//essa linha se aplica para os 2
//significa que passou a fila toda e nao encontrou onde largar entao provavelmente deu problema
IF i > 10 THEN
	xLimpaFilaTAG := TRUE;
END_IF

//limpa a fila de TAG
IF xLimpaFilaTAG THEN
	xLimpaFilaTAG := FALSE;
	FOR i := 0 TO 10 DO
		iFilaTAG[i] := 0;
	END_FOR
END_IF
END_ACTION

END_FUNCTION_BLOCK

// POUs/Automatico/Aspercao/RFIDeBalanca/FB_RFIDBalancaEntrada
FUNCTION_BLOCK FB_RFIDBalancaEntrada
VAR_INPUT
	xChegou : BOOL;//sinal de que uma carcaça chegou
	
	rPeso : REAL;//peso que veio da balanca
	xNovoPeso : BOOL;//sinal de que veio um novo peso
	
	iTAG : INT;//tag que veio da leitor
	xNovaTAG : BOOL;//sinal de que veio um novo tag
	
	iCamaraSelecionada : INT;//camara selecionada
	stHoraAhora 	: TIMESTRUCT; //Hora atual 
	sProcesso : STRING;//GUID do processo atual da camara que ele selecionou
	xLimpaFilaPeso : BOOL;
	xLimpaFilaTAG : BOOL;
END_VAR
VAR_OUTPUT
	iFilaTAG : ARRAY[0..10] OF INT;//fila das tag
	rFilaPeso : ARRAY[0..10] OF REAL;//fila dos pesos
	
	xEsperandoBalanca : BOOL;//se ta esperando vim o peso da balanca
	xEsperandoRFID : BOOL;//se ta esperando vim o valor da tag
	
	rPesoSelecionado : REAL;//qual peso ele selecionou e vai mandar para o banco
	iTAGSelecionado : INT;//qual tag ele selecionou e vai mandar para o banco
	
	stBuffer : ARRAY[0..9] OF st_BufferTagBalanca;
	
END_VAR
VAR
	i : INT;
	j : INT;
	rtChegouPeso : R_TRIG;
	rtTiraPeso : R_TRIG;
	xTiraPeso : BOOL;
	rtChegouTAG : R_TRIG;
	rtTiraTAG : R_TRIG;
	xTiraTAG : BOOL;
	
	rtChegou : R_TRIG;
	
	iEstado : INT;
	
						
	sSB		  : FB_StringBuilder;
    fbPLCDBCmd    : FB_PLCDBCmdEvt(sNetID := '', tTimeout := T#5S);
    sCmd          : STRING (1000); 
    aPara         : ST_ExpParameter;
	sAux 		  : STRING;
	
	stTSAux 	  : TIMESTRUCT; //Hora atual 
	
	
	saAux : ARRAY[0..50] OF STRING(80);//para gerar os comandos
	
END_VAR



IF true THEN	

	ControlePeso();
	ControleTAG();
	
	
	rtChegou(CLK:= xNovaTAG OR xChegou, Q=> );
	
	
	CASE  iEstado OF 
		0://esperando chegar 
			IF rtChegou.Q THEN
				xEsperandoBalanca := TRUE;
				xEsperandoRFID := TRUE;
				iEstado := 1;
			END_IF
			
		1://chegou fica esperando ter alguma 
				
			xEsperandoRFID := iFilaTAG[0] = 0;
			xEsperandoBalanca := rFilaPeso[0] = 0;
			
			IF NOT xEsperandoRFID AND NOT xEsperandoBalanca THEN
				iEstado := 2;
				rPesoSelecionado := rFilaPeso[0];
				xTiraPeso := TRUE;
				xEsperandoBalanca := FALSE;
				
				iTAGSelecionado := iFilaTAG[0];
				xTiraTAG := TRUE;
				xEsperandoRFID := FALSE;
				
				iEstado := 2;
				
				//ajusta no buffer
				FOR i := 9 TO 1 BY -1 DO
					stBuffer[i] := stBuffer[i-1];
				END_FOR
				
				stBuffer[0].iTag := iTAGSelecionado;
				stBuffer[0].rPeso := rPesoSelecionado;
				
				
			END_IF
		
		2://manda pro banco esses valores
		
			FOR i:= 0 TO 50 DO
				saAux[i] := '';
			END_FOR
			
			saAux[0] := ('INSERT INTO `geral`.`rfid` (`TAG`, `Processo`, ');
			saAux[1] := ('`Camara`, `PesoQuente`, `HoraPesoQuente`) VALUES ($'');
			saAux[2] := (TO_STRING(iTAGSelecionado));
			saAux[3] := ('$', $'');
			saAux[4] := (TO_STRING(sProcesso));
			saAux[5] := ('$', $'');
			saAux[6] := (TO_STRING(iCamaraSelecionada));
			saAux[7] := ('$', $'');
			saAux[8] := (TO_STRING(rPesoSelecionado));
			saAux[9] := ('$', $'');
			saAux[10] := (TO_STRING(stHoraAhora.wYear));
			saAux[11] := ('-');
			saAux[13] := (TO_STRING(stHoraAhora.wMonth));
			saAux[14] := ('-');
			saAux[15] := (TO_STRING(stHoraAhora.wDay));
			saAux[16] := (' ');
			saAux[17] := (TO_STRING(stHoraAhora.wHour));
			saAux[18] := (':');
			saAux[19] := (TO_STRING(stHoraAhora.wMinute));
			saAux[20] := (':');
			saAux[21] := (TO_STRING(stHoraAhora.wSecond));
			saAux[22] := ('$');');
			
			sCmd := F_ConcatArray1000(sArray:= saAux);
			
			aPara.eParaType := E_ExpParameterType.STRING_;
			aPara.nParaSize := SIZEOF(sAux);
		
			// call functionblock
			IF fbPLCDBCmd.Execute(
				hDBID:= 1, 
				pExpression:= ADR(sCmd), 
				cbExpression:= SIZEOF(sCmd), 
				pData:= ADR(sAux), 
				cbData:= SIZEOF(sAux), 
				pParameter:= ADR(aPara), 
				cbParameter:= SIZEOF(aPara)) 
			THEN
				iEstado := 0;
			END_IF
		
	END_CASE
	


END_IF

ACTION ControlePeso:



//Sobe na fila
rtChegouPeso(CLK:= xNovoPeso AND xEsperandoBalanca, Q=> );
IF rtChegouPeso.q THEN
	FOR i := 0 TO 9 DO
		IF rFilaPeso[i] = 0 THEN
			rFilaPeso[i] := rPeso;
			EXIT;
		END_IF
	END_FOR
END_IF


//Sobe na fila
rtTiraPeso(CLK:= xTiraPeso, Q=> );
IF rtTiraPeso.q THEN
	xTiraPeso := false;
	FOR i := 0 TO 9 DO
		IF rFilaPeso[i] = 0 THEN
			FOR j := 0 TO i DO
				rFilaPeso[j] := rFilaPeso[j+1];
			END_FOR
			EXIT;
		END_IF
	END_FOR
END_IF

//essa linha se aplica para os 2
//significa que passou a fila toda e nao encontrou onde largar entao provavelmente deu problema
IF i > 10 THEN
	xLimpaFilaPeso := TRUE;
END_IF

//limpa a fila de peso
IF xLimpaFilaPeso THEN
	xLimpaFilaPeso := FALSE;
	FOR i := 0 TO 10 DO
		rFilaPeso[i] := 0;
	END_FOR
END_IF
END_ACTION

ACTION ControleTAG:


//Sobe na fila
rtChegouTAG(CLK:= xNovaTAG, Q=> );
IF rtChegouTAG.q THEN
	FOR i := 0 TO 9 DO
		IF iFilaTAG[i] = 0 THEN
			iFilaTAG[i] := iTAG;
			EXIT;
		END_IF
	END_FOR
END_IF


//Sobe na fila
rtTiraTAG(CLK:= xTiraTAG, Q=> );
IF rtTiraTAG.q THEN
	xTiraTAG := false;
	FOR i := 0 TO 9 DO
		IF iFilaTAG[i] = 0 THEN
			FOR j := 0 TO i DO
				iFilaTAG[j] := iFilaTAG[j+1];
			END_FOR
			EXIT;
		END_IF
	END_FOR
END_IF

//essa linha se aplica para os 2
//significa que passou a fila toda e nao encontrou onde largar entao provavelmente deu problema
IF i > 10 THEN
	xLimpaFilaTAG := TRUE;
END_IF

//limpa a fila de TAG
IF xLimpaFilaTAG THEN
	xLimpaFilaTAG := FALSE;
	FOR i := 0 TO 10 DO
		iFilaTAG[i] := 0;
	END_FOR
END_IF
END_ACTION

END_FUNCTION_BLOCK

// POUs/Automatico/Aspercao/RFIDeBalanca/FB_RFIDBalancaSaida
FUNCTION_BLOCK FB_RFIDBalancaSaida
VAR_INPUT
	xChegou : BOOL;
	
	rPeso : REAL;
	xNovoPeso : BOOL;
	
	iTAG : INT;
	xNovaTAG : BOOL;
	
	iCamaraSelecionada : INT;
	stHoraAhora 	: TIMESTRUCT; //Hora atual 
	sProcesso : STRING;
	xLimpaFilaPeso : BOOL;
	xLimpaFilaTAG : BOOL;
	
END_VAR
VAR_OUTPUT
	iFilaTAG : ARRAY[0..10] OF INT;
	rFilaPeso : ARRAY[0..10] OF REAL;
	
	xEsperandoBalanca : BOOL;
	xEsperandoRFID : BOOL;
	
	rPesoSelecionado : REAL;
	iTAGSelecionado : INT;
	
	
	stBuffer : ARRAY[0..9] OF st_BufferTagBalanca;
	
END_VAR
VAR
	i : INT;
	j : INT;
	rtChegouPeso : R_TRIG;
	rtTiraPeso : R_TRIG;
	xTiraPeso : BOOL;
	rtChegouTAG : R_TRIG;
	rtTiraTAG : R_TRIG;
	xTiraTAG : BOOL;
	
	rtChegou : R_TRIG;
	
	iEstado : INT;
	
						
	//sSB		  : FB_StringBuilder;
    fbPLCDBCmd    : FB_PLCDBCmdEvt(sNetID := '', tTimeout := T#5S);
    sCmd          : STRING (1000); 
    aPara         : ST_ExpParameter;
	sAux 		  : STRING;
	
	stTSAux 	  : TIMESTRUCT; //Hora atual 
	
	saAux : ARRAY[0..50] OF STRING(80);//para gerar os comandos
	
	
END_VAR



IF true THEN	

	ControlePeso();
	ControleTAG();
	
	
	rtChegou(CLK:= xNovaTAG OR xChegou, Q=> );
	
	CASE  iEstado OF 
		0://esperando chegar 
			IF rtChegou.q THEN
				xEsperandoBalanca := TRUE;
				xEsperandoRFID := TRUE;
				iEstado := 1;
			END_IF
			
		1://chegou fica esperando ter alguma 
				
			xEsperandoRFID := iFilaTAG[0] = 0;
			xEsperandoBalanca := rFilaPeso[0] = 0;
			
			IF NOT xEsperandoRFID AND NOT xEsperandoBalanca THEN
				iEstado := 2;
				rPesoSelecionado := rFilaPeso[0];
				xTiraPeso := TRUE;
				xEsperandoBalanca := FALSE;
				
				iTAGSelecionado := iFilaTAG[0];
				xTiraTAG := TRUE;
				xEsperandoRFID := FALSE;
				
				iEstado := 2;
				
				//ajusta no buffer
				FOR i := 9 TO 1 BY -1 DO
					stBuffer[i] := stBuffer[i-1];
				END_FOR
				
				stBuffer[0].iTag := iTAGSelecionado;
				stBuffer[0].rPeso := rPesoSelecionado;
				
				
			END_IF
		
		2://manda pro banco esses valores
			//UPDATE `geral`.`rfid` SET `PesoFrio` = '12', `HoraPesoFrio` = 'xxx' WHERE (`TAG` = '12' and `Processo` = '{28F6E224-5F99-464E-8EF2-4966F1D308DE}');
			
			FOR i:= 0 TO 50 DO
				saAux[i] := '';
			END_FOR
			
			saAux[0] := ('UPDATE `geral`.`rfid` SET `PesoFrio` = $'');
			saAux[1] := (TO_STRING(rPesoSelecionado));
			saAux[2] := ('$', `Camara` = $'');
			saAux[3] := (TO_STRING(iCamaraSelecionada));
			saAux[4] := ('$', `HoraPesoFrio` = $'');
			saAux[5] := (TO_STRING(stHoraAhora.wYear));
			saAux[6] := ('-');
			saAux[7] := (TO_STRING(stHoraAhora.wMonth));
			saAux[8] := ('-');
			saAux[9] := (TO_STRING(stHoraAhora.wDay));
			saAux[10] := (' ');
			saAux[11] := (TO_STRING(stHoraAhora.wHour));
			saAux[12] := (':');
			saAux[13] := (TO_STRING(stHoraAhora.wMinute));
			saAux[14] := (':');
			saAux[15] := (TO_STRING(stHoraAhora.wSecond));
			saAux[16] := ('$' WHERE (`TAG` = $'');
			saAux[17] := (TO_STRING(iTAG));
			saAux[18] := ('$' and `PesoFrio` = $'');
			saAux[19] := ('-1');
			saAux[20] := ('$'');
			saAux[21] := ('');
			saAux[22] := (') ORDER BY id DESC LIMIT 1;');
			// PesoFrio` = '-1' and DATE(`HoraPesoQuente`) = DATE(DATE_ADD(now(), INTERVAL -1 DAY))) ORDER BY id DESC LIMIT 1;
			
			sCmd := F_ConcatArray1000(sArray:= saAux);
			
			aPara.eParaType := E_ExpParameterType.STRING_;
			aPara.nParaSize := SIZEOF(sAux);
		
			// call functionblock
			IF fbPLCDBCmd.Execute(
				hDBID:= 1, 
				pExpression:= ADR(sCmd), 
				cbExpression:= SIZEOF(sCmd), 
				pData:= ADR(sAux), 
				cbData:= SIZEOF(sAux), 
				pParameter:= ADR(aPara), 
				cbParameter:= SIZEOF(aPara)) 
			THEN
				iEstado := 0;
			END_IF
		
	END_CASE
	
	
	
	



END_IF

ACTION ControlePeso:



//Sobe na fila
rtChegouPeso(CLK:= xNovoPeso AND xEsperandoBalanca, Q=> );
IF rtChegouPeso.q THEN
	FOR i := 0 TO 9 DO
		IF rFilaPeso[i] = 0 THEN
			rFilaPeso[i] := rPeso;
			EXIT;
		END_IF
	END_FOR
END_IF


//Sobe na fila
rtTiraPeso(CLK:= xTiraPeso, Q=> );
IF rtTiraPeso.q THEN
	xTiraPeso := false;
	FOR i := 0 TO 9 DO
		IF rFilaPeso[i] = 0 THEN
			FOR j := 0 TO i DO
				rFilaPeso[j] := rFilaPeso[j+1];
			END_FOR
			EXIT;
		END_IF
	END_FOR
END_IF

//essa linha se aplica para os 2
//significa que passou a fila toda e nao encontrou onde largar entao provavelmente deu problema
IF i > 10 THEN
	xLimpaFilaPeso := TRUE;
END_IF

//limpa a fila de peso
IF xLimpaFilaPeso THEN
	xLimpaFilaPeso := FALSE;
	FOR i := 0 TO 10 DO
		rFilaPeso[i] := 0;
	END_FOR
END_IF
END_ACTION

ACTION ControleTAG:


//Sobe na fila
rtChegouTAG(CLK:= xNovaTAG, Q=> );
IF rtChegouTAG.q THEN
	FOR i := 0 TO 9 DO
		IF iFilaTAG[i] = 0 THEN
			iFilaTAG[i] := iTAG;
			EXIT;
		END_IF
	END_FOR
END_IF


//Sobe na fila
rtTiraTAG(CLK:= xTiraTAG, Q=> );
IF rtTiraTAG.q THEN
	xTiraTAG := false;
	FOR i := 0 TO 9 DO
		IF iFilaTAG[i] = 0 THEN
			FOR j := 0 TO i DO
				iFilaTAG[j] := iFilaTAG[j+1];
			END_FOR
			EXIT;
		END_IF
	END_FOR
END_IF

//essa linha se aplica para os 2
//significa que passou a fila toda e nao encontrou onde largar entao provavelmente deu problema
IF i > 10 THEN
	xLimpaFilaTAG := TRUE;
END_IF

//limpa a fila de TAG
IF xLimpaFilaTAG THEN
	xLimpaFilaTAG := FALSE;
	FOR i := 0 TO 10 DO
		iFilaTAG[i] := 0;
	END_FOR
END_IF
END_ACTION

END_FUNCTION_BLOCK

// POUs/Automatico/ControlesPID/FB_PIDeGrafico
FUNCTION_BLOCK FB_PIDeGrafico
VAR_IN_OUT
	stPID : stControlePID;
END_VAR
VAR_OUTPUT
END_VAR
VAR
	PID : FB_CTRL_PID;
	tonTempoDeAmostragem : TON;
	i : INT;
END_VAR





stPID.PID.EN.fSetpointValue := stPID.Config.rSetpoint;//Setpoint
stPID.PID.EN.fActualValue;//Valor atual
stPID.PID.EN.fManSyncValue;//Valor em manual
IF stPID.xLigaInterno THEN
	stPID.PID.EN.eMode := eCTRL_MODE_ACTIVE;
ELSE
	stPID.PID.EN.eMode := eCTRL_MODE_PASSIVE;	
END_IF
IF stPID.xReset THEN
	stPID.PID.EN.eMode := eCTRL_MODE_RESET;
END_IF
//eCTRL_MODE_PASSIVE - The output or outputs of the function block are set to zero, but the internal states are retained.
//eCTRL_MODE_ACTIVE - The function block is executed in accordance with its description, and appropriate output values are calculated (normal operation).
//eCTRL_MODE_RESET - In this operation mode all internal states are reset and the error bit is cleared.
//eCTRL_MODE_MANUAL - The value of the input value fManSyncValue is provided at the output (manual operation).
//eCTRL_STATE_IDLE - The function block has successfully been reset, and is now waiting for selection of the operation mode.


stPID.PID.stParams.tTaskCycleTime := T#10MS;//Tempo igual ao da Task PID
stPID.PID.stParams.tCtrlCycleTime := T#50MS;//A cada quanto tempo vai rodar o bloco

stPID.PID.stParams.fKp;//Controller amplification / controller coefficient
stPID.PID.stParams.tTn;//Integral action time; if this is parameterized to T#0s, the I component is deactivated.
stPID.PID.stParams.tTv;//Derivative action time; if this is parameterized to T#0s, the D component is deactivated.
stPID.PID.stParams.tTd;//Damping time
IF stPID.xPressao THEN
	stPID.PID.stParams.fOutMaxLimit := 100;
	stPID.PID.stParams.fOutMinLimit := 0;
ELSE
	stPID.PID.stParams.fOutMaxLimit := 100;
	stPID.PID.stParams.fOutMinLimit := 0;	
END_IF

aPID();

IF stPID.xPressao THEN
	stPID.PID.SA.rSaida := SCALE_R(X := stPID.PID.SA.fOut,
											I_LO := 0,
											I_HI := 100,
											O_LO := stPID.PID.EN.rMinimo,
											O_HI := stPID.PID.EN.rMaximo);
ELSE								
	stPID.PID.SA.rSaida := SCALE_R(X := stPID.PID.SA.fOut,
									I_LO := 0,
									I_HI := 100,
									O_LO := 100,
									O_HI := 0);	
									
	IF stPID.PID.SA.rSaida < stPID.PID.EN.rMinimo  THEN
		stPID.PID.SA.rSaida := stPID.PID.EN.rMinimo;
	END_IF	
							
	IF stPID.PID.SA.rSaida > stPID.PID.EN.rMaximo  THEN
		stPID.PID.SA.rSaida := stPID.PID.EN.rMaximo;
	END_IF

																	
END_IF
stPID.PID.SA.fOut;//Output of the PID element
stPID.PID.SA.eState;//State of the function block
TextoStatus();
stPID.PID.SA.bError;//Becomes TRUE, as soon as an error occurs.
stPID.PID.SA.eErrorId;//Supplies the error number when the output bError is set.
TextoErro();




Grafico();

ACTION aPID:
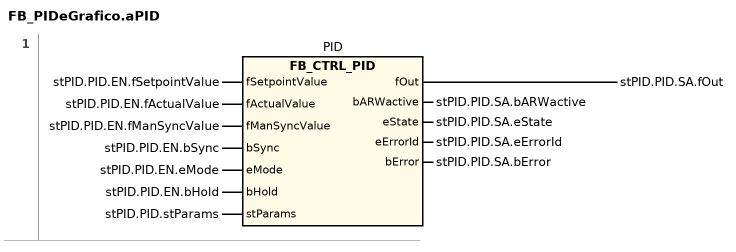
// NETWORK 1
PID(
    fSetpointValue := stPID.PID.EN.fSetpointValue,
    fActualValue := stPID.PID.EN.fActualValue,
    fManSyncValue := stPID.PID.EN.fManSyncValue,
    bSync := stPID.PID.EN.bSync,
    eMode := stPID.PID.EN.eMode,
    bHold := stPID.PID.EN.bHold,
    stParams := stPID.PID.stParams,
    bARWactive => stPID.PID.SA.bARWactive,
    eState => stPID.PID.SA.eState,
    eErrorId => stPID.PID.SA.eErrorId,
    bError => stPID.PID.SA.bError); // FB_CTRL_PID
stPID.PID.SA.fOut := PID.fOut;
END_ACTION

ACTION Grafico:


IF tonTempoDeAmostragem.q THEN
	tonTempoDeAmostragem(IN:= FALSE);
END_IF
tonTempoDeAmostragem(IN:= TRUE, PT:= T#0.5S, Q=> , ET=> );


IF tonTempoDeAmostragem.q THEN
	
	FOR I := 0 TO 119 BY 1 DO
		stPID.Grafico[0,i].y := stPID.Grafico[0,i+1].y ;
		stPID.Grafico[1,i].y := stPID.Grafico[1,i+1].y ;
		stPID.Grafico[2,i].y := stPID.Grafico[2,i+1].y ;
		stPID.Grafico[3,i].y := stPID.Grafico[3,i+1].y ;
		
		stPID.Grafico[0,i].x := TO_STRING(i);
		stPID.Grafico[0,i].sCor := '#007fad';
		stPID.Grafico[0,i].sTipo := 'line';
		stPID.Grafico[0,i].label := 'Setpoint';
		
		stPID.Grafico[1,i].x := TO_STRING(i);
		stPID.Grafico[1,i].sCor := '#c7ae0a';
		stPID.Grafico[1,i].sTipo := 'line';
		
		
	
		
		stPID.Grafico[2,i].x := TO_STRING(i);
		stPID.Grafico[2,i].sCor := '#2d0ac7';
		stPID.Grafico[2,i].sTipo := 'line';
		
	
		
		stPID.Grafico[3,i].x := TO_STRING(i);
		stPID.Grafico[3,i].sCor := '#FF0000';
		stPID.Grafico[3,i].sTipo := 'line';
		
		
		IF stPID.xPressao THEN
			stPID.Grafico[1,i].label := ' Bomba';
			stPID.Grafico[2,i].label := 'Pressao Fim';
			stPID.Grafico[3,i].label := 'Pressao Inicio';
		ELSE
			stPID.Grafico[1,i].label := ' Valvula';
			stPID.Grafico[2,i].label := 'Temperatura fim';
			stPID.Grafico[3,i].label := 'Temperatura Inicio';
		END_IF
	END_FOR
	
	stPID.Grafico[0,120] := stPID.Grafico[0,1];
	stPID.Grafico[1,120] := stPID.Grafico[1,1];
	stPID.Grafico[2,120] := stPID.Grafico[2,1];
	stPID.Grafico[3,120] := stPID.Grafico[3,1];
	
	stPID.Grafico[0,120].y := stPID.PID.EN.fSetpointValue;
	
	IF stPID.xPressao THEN
		stPID.Grafico[1,120].y := stPID.PID.SA.fOut/100;
	ELSE
		stPID.Grafico[1,120].y := stPID.PID.SA.fOut/10;		
	END_IF
	stPID.Grafico[2,120].y := stPID.PID.EN.fActualValue;
	stPID.Grafico[3,120].y := stPID.rOutraNoGrafico;
	
	
	
END_IF
END_ACTION

ACTION TextoErro:



CASE stPID.PID.SA.eErrorId OF
	
	 0: stPID.PID.SA.sErrorId := 'NOERROR';
	 1: stPID.PID.SA.sErrorId := 'INVALIDTASKCYCLETIME';
	 2: stPID.PID.SA.sErrorId := 'INVALIDCTRLCYCLETIME';
	 3: stPID.PID.SA.sErrorId := 'INVALIDPARAM';
	 4: stPID.PID.SA.sErrorId := 'INVALIDPARAM_Tv';
	 5: stPID.PID.SA.sErrorId := 'INVALIDPARAM_Td';
	 6: stPID.PID.SA.sErrorId := 'INVALIDPARAM_Tn';
	 7: stPID.PID.SA.sErrorId := 'INVALIDPARAM_Ti';
	 8: stPID.PID.SA.sErrorId := 'INVALIDPARAM_fHystereisisRange';
	 9: stPID.PID.SA.sErrorId := 'INVALIDPARAM_fPosOutOn_Off';
	 10: stPID.PID.SA.sErrorId := 'INVALIDPARAM_fNegOutOn_Off';
	 11: stPID.PID.SA.sErrorId := 'INVALIDPARAM_TableDescription';
	 12: stPID.PID.SA.sErrorId := 'INVALIDPARAM_TableData';
	 13: stPID.PID.SA.sErrorId := 'INVALIDPARAM_DataTableADR';
	 14: stPID.PID.SA.sErrorId := 'INVALIDPARAM_T0';
	 15: stPID.PID.SA.sErrorId := 'INVALIDPARAM_T1';
	 16: stPID.PID.SA.sErrorId := 'INVALIDPARAM_T2';
	 17: stPID.PID.SA.sErrorId := 'INVALIDPARAM_T3';
	 18: stPID.PID.SA.sErrorId := 'INVALIDPARAM_Theta';
	 19: stPID.PID.SA.sErrorId := 'INVALIDPARAM_nOrder';
	 20: stPID.PID.SA.sErrorId := 'INVALIDPARAM_Tt';
	 21: stPID.PID.SA.sErrorId := 'INVALIDPARAM_Tu';
	 22: stPID.PID.SA.sErrorId := 'INVALIDPARAM_Tg';
	 23: stPID.PID.SA.sErrorId := 'INVALIDPARAM_infinite_slope';
	 24: stPID.PID.SA.sErrorId := 'INVALIDPARAM_fMaxIsLessThanfMin';
	 25: stPID.PID.SA.sErrorId := 'INVALIDPARAM_fOutMaxLimitIsLessThanfOutMinLimit ';
	 26: stPID.PID.SA.sErrorId := 'INVALIDPARAM_fOuterWindow';
	 27: stPID.PID.SA.sErrorId := 'INVALIDPARAM_fInnerWindow';
	 28: stPID.PID.SA.sErrorId := 'INVALIDPARAM_fOuterWindowIsLessThanfInnerWindow ';
	 29: stPID.PID.SA.sErrorId := 'INVALIDPARAM_fDeadBandInput';
	 30: stPID.PID.SA.sErrorId := 'INVALIDPARAM_fDeadBandOutput';
	 31: stPID.PID.SA.sErrorId := 'INVALIDPARAM_PWM_Cycletime';
	 32: stPID.PID.SA.sErrorId := 'INVALIDPARAM_no_Parameterset';
	 33: stPID.PID.SA.sErrorId := 'INVALIDPARAM_fOutOn';
	 34: stPID.PID.SA.sErrorId := 'INVALIDPARAM_fOutOff';
	 35: stPID.PID.SA.sErrorId := 'INVALIDPARAM_fGain';
	 36: stPID.PID.SA.sErrorId := 'INVALIDPARAM_fOffset';
	 37: stPID.PID.SA.sErrorId := 'MODE_NOT_SUPPORTED';
	 38: stPID.PID.SA.sErrorId := 'INVALIDPARAM_Tv_heating';
	 39: stPID.PID.SA.sErrorId := 'INVALIDPARAM_Td_heating';
	 40: stPID.PID.SA.sErrorId := 'INVALIDPARAM_Tn_heating';
	 41: stPID.PID.SA.sErrorId := 'INVALIDPARAM_Tv_cooling';
	 42: stPID.PID.SA.sErrorId := 'INVALIDPARAM_Td_cooling';
	 43: stPID.PID.SA.sErrorId := 'INVALIDPARAM_Tn_cooling';
	 44: stPID.PID.SA.sErrorId := 'RANGE_NOT_SUPPORTED';
	 45: stPID.PID.SA.sErrorId := 'INVALIDPARAM_nParameterChangeCycleTicks';
	 46: stPID.PID.SA.sErrorId := 'ParameterEstimationFailed';
	 47: stPID.PID.SA.sErrorId := 'NoiseLevelToHigh';
	 48: stPID.PID.SA.sErrorId := 'INTERNAL_ERROR_0';
	 49: stPID.PID.SA.sErrorId := 'INTERNAL_ERROR_1';
	 50: stPID.PID.SA.sErrorId := 'INTERNAL_ERROR_2';
	 51: stPID.PID.SA.sErrorId := 'INTERNAL_ERROR_3';
	 52: stPID.PID.SA.sErrorId := 'INTERNAL_ERROR_4';
	 53: stPID.PID.SA.sErrorId := 'INTERNAL_ERROR_5';
	 54: stPID.PID.SA.sErrorId := 'INTERNAL_ERROR_6';
	 55: stPID.PID.SA.sErrorId := 'INTERNAL_ERROR_7';
	 56: stPID.PID.SA.sErrorId := 'INTERNAL_ERROR_8';
	 57: stPID.PID.SA.sErrorId := 'INTERNAL_ERROR_9';
	 58: stPID.PID.SA.sErrorId := 'INVALIDPARAM_WorkArrayADR';
	 59: stPID.PID.SA.sErrorId := 'INVALIDPARAM_tOnTiime';
	 60: stPID.PID.SA.sErrorId := 'INVALIDPARAM_tOffTiime';
	 61: stPID.PID.SA.sErrorId := 'INVALIDPARAM_nMaxMovingPulses';
	 62: stPID.PID.SA.sErrorId := 'INVALIDPARAM_nAdditionalPulsesAtLimits';
	 63: stPID.PID.SA.sErrorId := 'INVALIDPARAM_fCtrlOutMax_Min';
	 64: stPID.PID.SA.sErrorId := 'INVALIDPARAM_fDeltaMax';
	 65: stPID.PID.SA.sErrorId := 'INVALIDPARAM_tMovingTime';
	 66: stPID.PID.SA.sErrorId := 'INVALIDPARAM_tDeadTime';
	 67: stPID.PID.SA.sErrorId := 'INVALIDPARAM_tAdditionalMoveTimeAtLimits';
	 68: stPID.PID.SA.sErrorId := 'INVALIDPARAM_fThreshold';
	 69: stPID.PID.SA.sErrorId := 'MEMCPY';
	 70: stPID.PID.SA.sErrorId := 'MEMSET';
	 71: stPID.PID.SA.sErrorId := 'INVALIDPARAM_nNumberOfColumns';
	 72: stPID.PID.SA.sErrorId := 'FileClose';
	 73: stPID.PID.SA.sErrorId := 'FileOpen';
	 74: stPID.PID.SA.sErrorId := 'FileWrite';
	 75: stPID.PID.SA.sErrorId := 'INVALIDPARAM_fVeloNeg';
	 76: stPID.PID.SA.sErrorId := 'INVALIDPARAM_fVeloPos';
	 77: stPID.PID.SA.sErrorId := 'INVALIDPARAM_DeadBandInput';
	 78: stPID.PID.SA.sErrorId := 'INVALIDPARAM_DeadBandOutput';
	 79: stPID.PID.SA.sErrorId := 'INVALIDPARAM_CycleDuration';
	 80: stPID.PID.SA.sErrorId := '  INVALIDPARAM_tStart';
	 81: stPID.PID.SA.sErrorId := 'INVALIDPARAM_StepHeigthTuningToLow';
	 82: stPID.PID.SA.sErrorId := 'INVALIDPARAM_fMinLimitIsLessThanZero';
	 83: stPID.PID.SA.sErrorId := 'INVALIDPARAM_fMaxLimitIsGreaterThan100';
	 84: stPID.PID.SA.sErrorId := 'INVALIDPARAM_fStepSize';
	 85: stPID.PID.SA.sErrorId := 'INVALIDPARAM_fOkRangeIsLessOrEqualZero';
	 86: stPID.PID.SA.sErrorId := 'INVALIDPARAM_fForceRangeIsLessOrEqualfOkRange ';
	 87: stPID.PID.SA.sErrorId := 'INVALIDPWMPeriod';
	 88: stPID.PID.SA.sErrorId := 'INVALIDPARAM_tMinimumPulseTime';
	 89: stPID.PID.SA.sErrorId := 'FileDelete';
	 90: stPID.PID.SA.sErrorId := 'INVALIDPARAM_nNumberOfPwmOutputs';
	 91: stPID.PID.SA.sErrorId := 'INVALIDPARAM_nPwmInputArray_SIZEOF';
	 92: stPID.PID.SA.sErrorId := 'INVALIDPARAM_nPwmOutputArray_SIZEOF';
	 93: stPID.PID.SA.sErrorId := 'INVALIDPARAM_nPwmWaitTimesConfig_SIZEOF';
	 94: stPID.PID.SA.sErrorId := 'INVALIDPARAM_nPwmInternalData_SIZEOF';
	 95: stPID.PID.SA.sErrorId := 'SIZEOF';
	 96: stPID.PID.SA.sErrorId := 'INVALIDPARAM_nOrderOfTheTransferfunction';
	 97: stPID.PID.SA.sErrorId := 'INVALIDPARAM_nNumeratorArray_SIZEOF';
	 98: stPID.PID.SA.sErrorId := 'INVALIDPARAM_nDenominatorArray_SIZEOF';
	 99: stPID.PID.SA.sErrorId := 'INVALIDPARAM_a_n_IsZero';
	 100: stPID.PID.SA.sErrorId := 'INVALIDPARAM_WorkArraySIZEOF';
	 101: stPID.PID.SA.sErrorId := 'INVALIDPARAM_MOVINGRANGE_MIN_MAX';
	 102: stPID.PID.SA.sErrorId := 'INVALIDPARAM_MOVINGTIME';
	 103: stPID.PID.SA.sErrorId := 'INVALIDPARAM_DEADTIME';
	 104: stPID.PID.SA.sErrorId := 'INVALIDPARAM_fMinLimitIsGreaterThanfMaxLimit';
	 105: stPID.PID.SA.sErrorId := 'INVALIDPARAM_DataTableSIZEOF';
	 106: stPID.PID.SA.sErrorId := 'INVALIDPARAM_OutputVectorDescription';
	 107: stPID.PID.SA.sErrorId := 'TaskCycleTimeChanged';
	 108: stPID.PID.SA.sErrorId := 'INVALIDPARAM_nMinMovingPulses';
	 109: stPID.PID.SA.sErrorId := 'INVALIDPARAM_fAcceleration';
	 110: stPID.PID.SA.sErrorId := 'INVALIDPARAM_fDeceleration';
	 111: stPID.PID.SA.sErrorId := 'INVALIDPARAM_StartAndTargetPos';
	 112: stPID.PID.SA.sErrorId := 'INVALIDPARAM_fVelocity';
	 113: stPID.PID.SA.sErrorId := 'INVALIDPARAM_fTargetPos';
	 114: stPID.PID.SA.sErrorId := 'INVALIDPARAM_fStartPos';
	 115: stPID.PID.SA.sErrorId := 'INVALIDPARAM_fMovingLength';
	 116: stPID.PID.SA.sErrorId := 'NT_GetTime';
	 117: stPID.PID.SA.sErrorId := 'INVALIDPARAM_No3PhaseSolutionPossible';
	 118: stPID.PID.SA.sErrorId := 'INVALIDPARAM_fStartVelo';
	 119: stPID.PID.SA.sErrorId := 'INVALIDPARAM_fTargetVelo';
	 120: stPID.PID.SA.sErrorId := 'INVALID_NEW_PARAMETER_TYPE';
	 121: stPID.PID.SA.sErrorId := 'INVALIDPARAM_fBaseTime';
	 122: stPID.PID.SA.sErrorId := 'INVALIDPARAM_nOrderOfTheTransferfunction_SIZEOF ';
	 124: stPID.PID.SA.sErrorId := 'INVALIDPARAM_nFilterOrder';
	 125: stPID.PID.SA.sErrorId := 'INVALIDPARAM_nCoefficientsArray_a_SIZEOF';
	 126: stPID.PID.SA.sErrorId := 'INVALIDPARAM_nCoefficientsArray_b_SIZEOF';
	 127: stPID.PID.SA.sErrorId := 'INVALIDPARAM_nDigitalFiterData_SIZEOF';
	 128: stPID.PID.SA.sErrorId := 'INVALIDPARAM_nLogBuffer_SIZEOF';
	 129: stPID.PID.SA.sErrorId := 'LogBufferOverflow';
	 130: stPID.PID.SA.sErrorId := 'INVALIDPARAM_nLogBuffer_ADR';
	 131: stPID.PID.SA.sErrorId := 'INVALIDPARAM_nCoefficientsArray_a_ADR';
	 132: stPID.PID.SA.sErrorId := 'INVALIDPARAM_nCoefficientsArray_b_ADR';
	 133: stPID.PID.SA.sErrorId := 'INVALIDPARAM_nPwmInputArray_ADR';
	 134: stPID.PID.SA.sErrorId := 'INVALIDPARAM_nPwmOutputArray_ADR';
	 135: stPID.PID.SA.sErrorId := 'INVALIDPARAM_nPwmWaitTimesConfig_ADR';
	 136: stPID.PID.SA.sErrorId := 'INVALIDPARAM_nPwmInternalData_ADR';
	 137: stPID.PID.SA.sErrorId := 'INVALIDPARAM_nDigitalFiterData_ADR';
	 138: stPID.PID.SA.sErrorId := 'INVALIDPARAM_nNumeratorArray_ADR';
	 139: stPID.PID.SA.sErrorId := 'INVALIDPARAM_nDenominatorArray_ADR';
	 140: stPID.PID.SA.sErrorId := 'INVALIDPARAM_nTransferfunction1Data_ADR';
	 141: stPID.PID.SA.sErrorId := 'INVALIDPARAM_nTransferfunction2Data_ADR';
	 142: stPID.PID.SA.sErrorId := 'FileSeek';
	 143: stPID.PID.SA.sErrorId := 'INVALIDPARAM_AmbientTempMaxIsLessThanAmbientTempMin';
	 144: stPID.PID.SA.sErrorId := 'INVALIDPARAM_ForerunTempMaxIsLessThanForerunTempMin';
	 145: stPID.PID.SA.sErrorId := 'INVALIDLOGCYCLETIME';
	 146: stPID.PID.SA.sErrorId := 'INVALIDVERSION_TcControllerToolbox';
	 147: stPID.PID.SA.sErrorId := 'INVALIDPARAM_Bandwidth';
	 148: stPID.PID.SA.sErrorId := 'INVALIDPARAM_NotchFrequency';
	 149: stPID.PID.SA.sErrorId := 'INVALIDPARAM_DampingCoefficient';
	 150: stPID.PID.SA.sErrorId := 'INVALIDPARAM_fKpIsLessThanZero';
 
END_CASE
END_ACTION

ACTION TextoStatus:







CASE stPID.PID.SA.eState OF 
	0: stPID.PID.SA.sState := 'IDLE';
	1: stPID.PID.SA.sState := 'PASSIVE';
	2: stPID.PID.SA.sState := 'ACTIVE';
	3: stPID.PID.SA.sState := 'RESET';
	4: stPID.PID.SA.sState := 'MANUAL';
	5: stPID.PID.SA.sState := 'TUNING';
	6: stPID.PID.SA.sState := 'TUNED';
	7: stPID.PID.SA.sState := 'SELFTEST';
	8: stPID.PID.SA.sState := 'ERROR';
	9: stPID.PID.SA.sState := 'SYNC_MOVEMENT';
END_CASE
END_ACTION

END_FUNCTION_BLOCK

// POUs/MAIN
PROGRAM MAIN
VAR
	

	fb1 : FB_Balanca;
	fb2 : FB_SalvaBalancaBanco;
	fb3 : FB_Camaras;
	fb4 : FB_SalvaEventoRelatorio;
	fb5 : FB_ControleSaidaAreaFria;
	fb6 : FB_ControleEntradaAreaQuente;
	fb7 : FB_ControleEdicaoProtocolo;
	fb8 : FB_ControleValvulaApersao;
	fb9 : FB_PIDeGrafico;



END_VAR

END_PROGRAM

// POUs/ValidaLicensa
PROGRAM ValidaLicensa
VAR
{attribute 'tc_no_symbol'}
Olhaliscensa : FB_CheckLicense;
{attribute 'tc_no_symbol'}
GUIDLicensa : GUID := STRING_TO_GUID('0A869185-D298-45F0-9D7B-88C4360BE2C8');
END_VAR


Licensas();

STCheckLicense := Olhaliscensa.stCheckLicense;

xLicensaValida6446896834 :=
 Olhaliscensa.stCheckLicense.eResult = 0 OR
 Olhaliscensa.stCheckLicense.eResult = 16#203 OR
 Olhaliscensa.stCheckLicense.eResult = 16#254 OR
 Olhaliscensa.stCheckLicense.eResult = 16#255;

 LicensaValida := xLicensaValida6446896834;

ACTION Licensas:
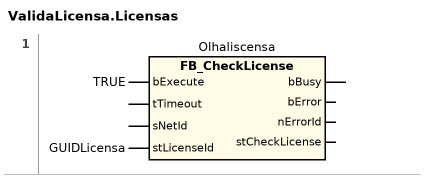
// NETWORK 1
Olhaliscensa(bExecute := TRUE, stLicenseId := GUIDLicensa); // FB_CheckLicense
END_ACTION

END_PROGRAM
